Omron Sysmac Studio project BaskiMakinesi_Uygulamasi (Sysmac Studio 1.65.0.64007, StandardProject)

# Controller new_Controller_0: NX1P2-1040DT1 version 1.69
Task PrimaryTask (priority 4, period or condition 2000): Program0

VAR_GLOBAL
    IN_Start_Buton : BOOL;
    IN_Stop_Buton : BOOL;
    IN_ACS_Buton : BOOL;
    IN_UrunAlgilama_Sens : BOOL;
    OUT_Konveyor_Start : BOOL;
    OUT_Valf1 : BOOL;
    OUT_Valf2 : BOOL;
    OUT_Baski_Valfi : BOOL;
    OUT_Valf3 : BOOL;
    OUT_Valf4 : BOOL;
END_VAR

PROGRAM Program0
VAR
    SistemStart : BOOL;
    Adim : INT;
    Adiim : INT;
    TON_Valf_1 : TON;
    TON_Valf_2 : TON;
    TON_Valf_3 : TON;
    TON_Valf_4 : TON;
    TON_Konveyor_Delay : TON;
END_VAR
VAR_EXTERNAL
    IN_Start_Buton : BOOL;
    IN_Stop_Buton : BOOL;
    IN_ACS_Buton : BOOL;
    IN_UrunAlgilama_Sens : BOOL;
    OUT_Konveyor_Start : BOOL;
    OUT_Valf1 : BOOL;
    OUT_Valf3 : BOOL;
    OUT_Valf2 : BOOL;
    OUT_Valf4 : BOOL;
END_VAR

(* Section Section0: ladder, written here as Structured Text *)

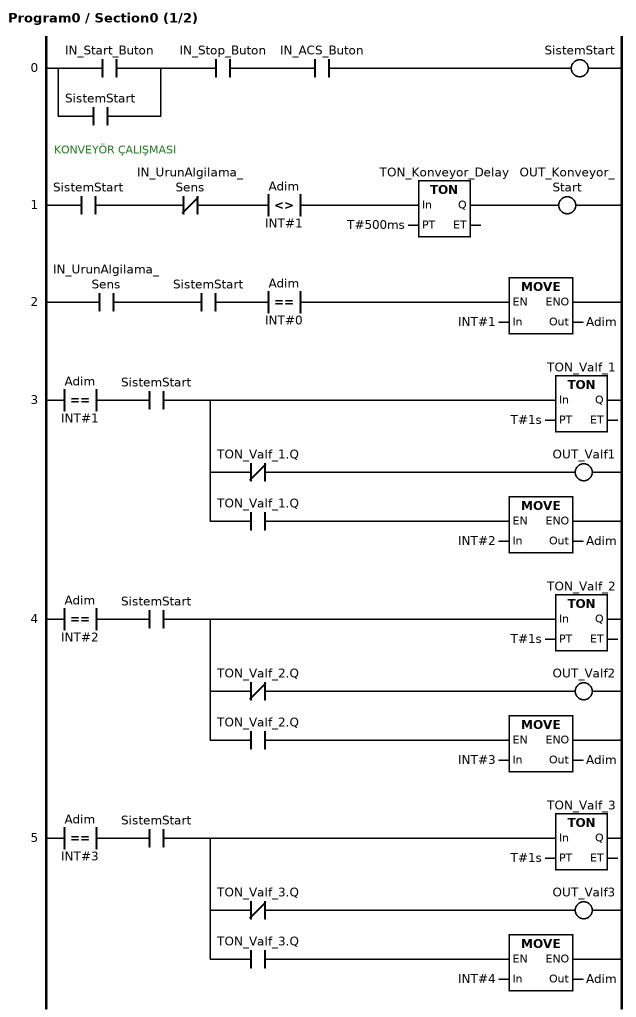
(* Rung 0 *)
SistemStart := (IN_Start_Buton OR SistemStart) AND IN_Stop_Buton AND IN_ACS_Buton;
(* Rung 1: KONVEYÖR ÇALIŞMASI *)
TON_Konveyor_Delay(In := SistemStart AND NOT IN_UrunAlgilama_Sens AND (Adim <> INT#1), PT := T#500ms);
OUT_Konveyor_Start := TON_Konveyor_Delay.Q;
(* Rung 2 *)
IF IN_UrunAlgilama_Sens AND SistemStart AND (Adim = INT#0) THEN Adim := INT#1; END_IF;
(* Rung 3 *)
TON_Valf_1(In := (Adim = INT#1) AND SistemStart, PT := T#1s);
OUT_Valf1 := (Adim = INT#1) AND SistemStart AND NOT TON_Valf_1.Q;
IF (Adim = INT#1) AND SistemStart AND TON_Valf_1.Q THEN Adim := INT#2; END_IF;
(* Rung 4 *)
TON_Valf_2(In := (Adim = INT#2) AND SistemStart, PT := T#1s);
OUT_Valf2 := (Adim = INT#2) AND SistemStart AND NOT TON_Valf_2.Q;
IF (Adim = INT#2) AND SistemStart AND TON_Valf_2.Q THEN Adim := INT#3; END_IF;
(* Rung 5 *)
TON_Valf_3(In := (Adim = INT#3) AND SistemStart, PT := T#1s);
OUT_Valf3 := (Adim = INT#3) AND SistemStart AND NOT TON_Valf_3.Q;
IF (Adim = INT#3) AND SistemStart AND TON_Valf_3.Q THEN Adim := INT#4; END_IF;

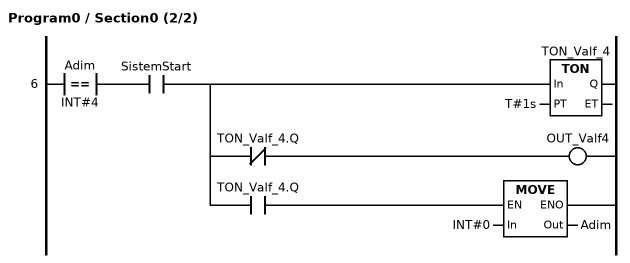
(* Rung 6 *)
TON_Valf_4(In := (Adim = INT#4) AND SistemStart, PT := T#1s);
OUT_Valf4 := (Adim = INT#4) AND SistemStart AND NOT TON_Valf_4.Q;
IF (Adim = INT#4) AND SistemStart AND TON_Valf_4.Q THEN Adim := INT#0; END_IF;
END_PROGRAM